FUNCTION HYP : lreal
VAR_INPUT
	X :LREAL;
	Y :LREAL;
END_VAR
VAR
END_VAR

HYP := sqrt(expt(X,2)+expt(Y,2));

END_FUNCTION

(* stored: Version 1.1.0.1, ProductVersion 3.1.4024.11
   POU HYP: Id {c1201563-527e-4793-9258-0d9f4500e7b3}, SpecialFunc None *)
